Staubli VAL3: __ts_english.pgx

program __ts_english()
begin
  //
end
